FUNCTION FILLSTRING : STRING
VAR_INPUT
	str : STRING;
	strlen : INT;
	fill_char : STRING(1);
END_VAR
VAR
	rawlen : INT;
	
	fillNumber : INT;
	
	tmpstr : STRING;
	
	i : INT;
END_VAR

rawlen := LEN(STR:= str);

fillNumber := strlen - rawlen;

tmpstr := '';

FOR i:= 1 TO fillNumber DO
	tmpstr := CONCAT(STR1:= tmpstr, STR2:= fill_char);
END_FOR

FILLSTRING := CONCAT(STR1:= tmpstr, STR2:= str);

END_FUNCTION

(* stored: Version 1.1.0.1, ProductVersion 3.1.4026.13
   POU FILLSTRING: Id {1813ba20-26f0-40fc-8701-d599c7075920}, SpecialFunc None *)
